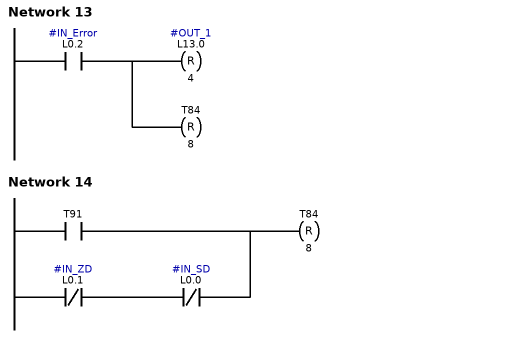
[picture p192: SBR88 networks 13-14]
Network 13
LD     #IN_Error:L0.2
R      #OUT_1:L13.0, 4
R      T84, 8
Network 14
LD     T91
LDN    #IN_ZD:L0.1
AN     #IN_SD:L0.0
OLD
R      T84, 8
END_SUBROUTINE_BLOCK

SUBROUTINE_BLOCK 除铁器4组5:SBR89
TITLE=
VAR_INPUT
IN_SD:BOOL;	// L0.0 
IN_ZD:BOOL;	// L0.1 
IN_Error:BOOL;	// L0.2 
IN_Run_Time:INT;	// LW1 
IN_Stop_Time:INT;	// LW3 
Z_Time:DINT;	// LD5 
END_VAR
VAR_IN_OUT
JS:DINT;	// LD9 
END_VAR
VAR_OUTPUT
OUT_1:BOOL;	// L13.0 
OUT_2:BOOL;	// L13.1 
OUT_3:BOOL;	// L13.2 
OUT_4:BOOL;	// L13.3 
END_VAR
VAR
TP1:BOOL;	// L13.4 
TP2:BOOL;	// L13.5 
END_VAR
BEGIN
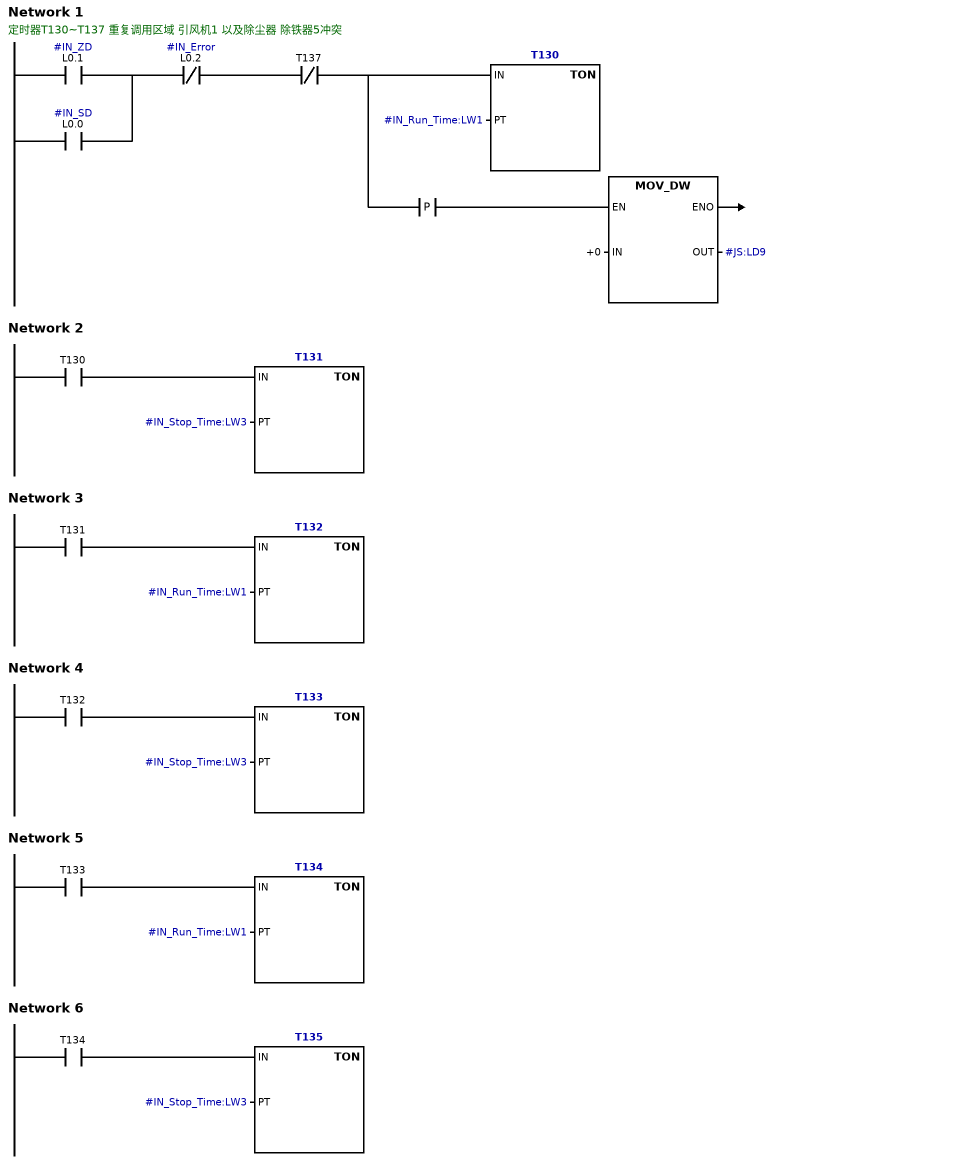
Network 1
// 定时器T130~T137 重复调用区域 引风机1 以及除尘器 除铁器5冲突
LD     #IN_ZD:L0.1
O      #IN_SD:L0.0
AN     #IN_Error:L0.2
AN     T137
TON    T130, #IN_Run_Time:LW1
EU
MOVD   +0, #JS:LD9
Network 2
LD     T130
TON    T131, #IN_Stop_Time:LW3
Network 3
LD     T131
TON    T132, #IN_Run_Time:LW1
Network 4
LD     T132
TON    T133, #IN_Stop_Time:LW3
Network 5
LD     T133
TON    T134, #IN_Run_Time:LW1
Network 6
LD     T134
TON    T135, #IN_Stop_Time:LW3
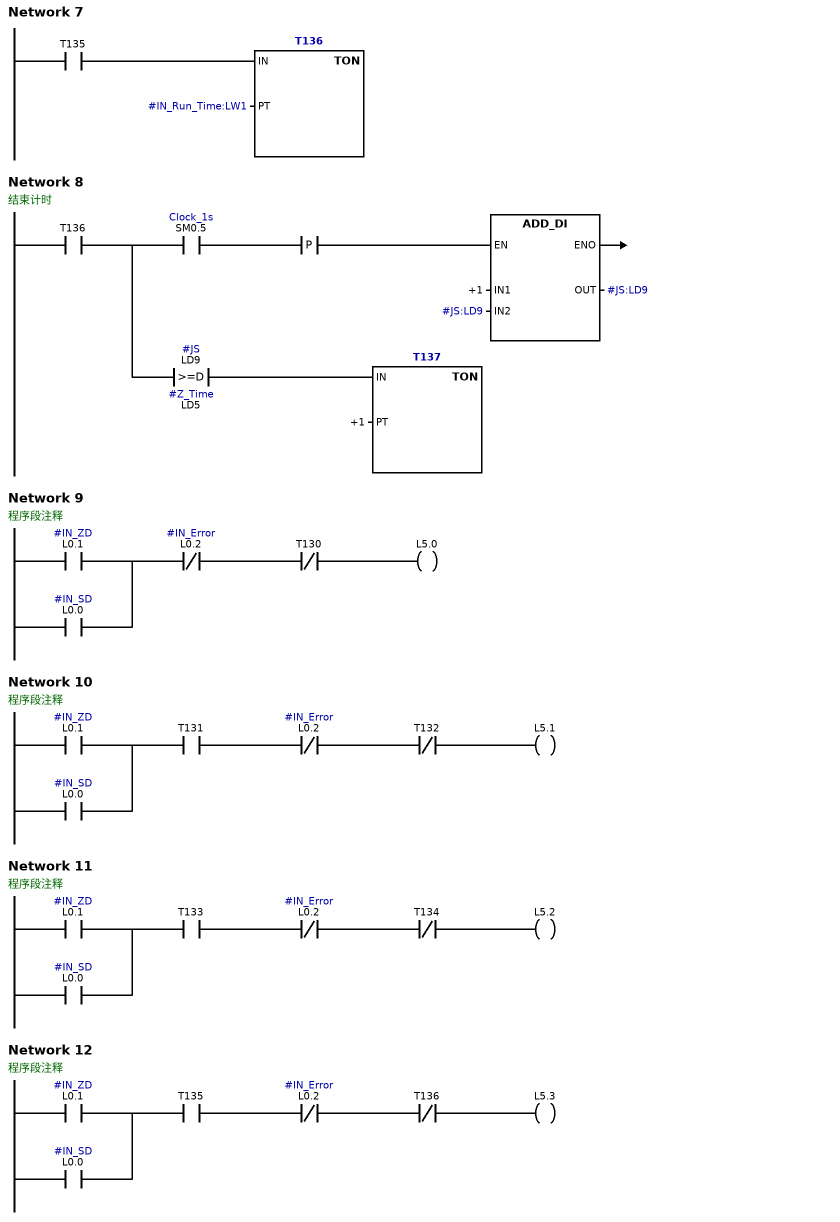
Network 7
LD     T135
TON    T136, #IN_Run_Time:LW1
Network 8
// 结束计时
LD     T136
LPS
A      Clock_1s:SM0.5
EU
+D     +1, #JS:LD9
LPP
AD>=   #JS:LD9, #Z_Time:LD5
TON    T137, +1
Network 9
//  程序段注释
LD     #IN_ZD:L0.1
O      #IN_SD:L0.0
AN     #IN_Error:L0.2
AN     T130
=      L5.0
Network 10
//  程序段注释
LD     #IN_ZD:L0.1
O      #IN_SD:L0.0
A      T131
AN     #IN_Error:L0.2
AN     T132
=      L5.1
Network 11
//  程序段注释
LD     #IN_ZD:L0.1
O      #IN_SD:L0.0
A      T133
AN     #IN_Error:L0.2
AN     T134
=      L5.2
Network 12
//  程序段注释
LD     #IN_ZD:L0.1
O      #IN_SD:L0.0
A      T135
AN     #IN_Error:L0.2
AN     T136
=      L5.3
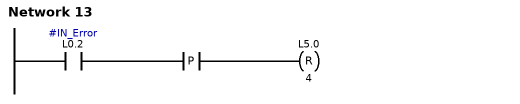
Network 13
LD     #IN_Error:L0.2
EU
R      L5.0, 4
END_SUBROUTINE_BLOCK

SUBROUTINE_BLOCK 膨胀阀4组1:SBR90
TITLE=
VAR_INPUT
IN_SD:BOOL;	// L0.0 
IN_ZD:BOOL;	// L0.1 
IN_Error:BOOL;	// L0.2 
IN_Run_Time:INT;	// LW1 
IN_Stop_Time:INT;	// LW3 
END_VAR
VAR_OUTPUT
OUT_1:BOOL;	// L5.0 膨胀1
OUT_2:BOOL;	// L5.1 下料1
OUT_3:BOOL;	// L5.2 膨胀2
OUT_4:BOOL;	// L5.3 下料2
END_VAR
VAR
TP1:BOOL;	// L5.4 
TP2:BOOL;	// L5.5 
END_VAR
BEGIN
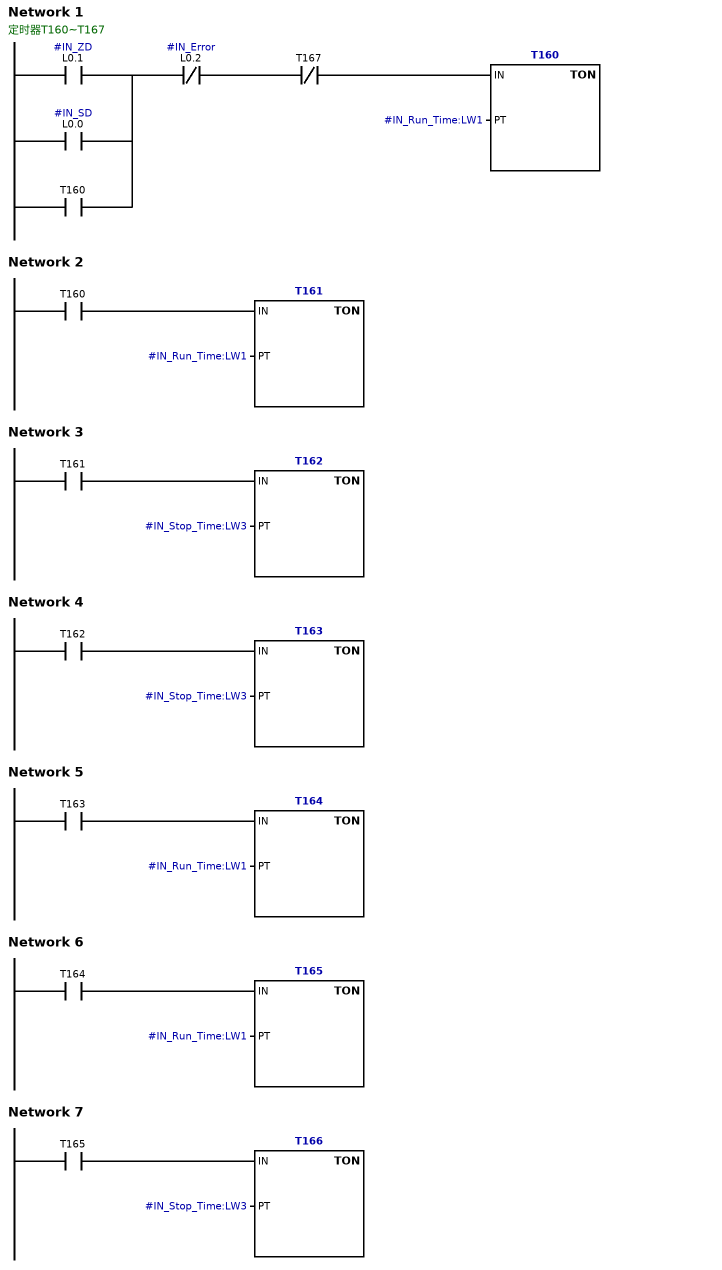
Network 1
// 定时器T160~T167
LD     #IN_ZD:L0.1
O      #IN_SD:L0.0
O      T160
AN     #IN_Error:L0.2
AN     T167
TON    T160, #IN_Run_Time:LW1
Network 2
LD     T160
TON    T161, #IN_Run_Time:LW1
Network 3
LD     T161
TON    T162, #IN_Stop_Time:LW3
Network 4
LD     T162
TON    T163, #IN_Stop_Time:LW3
Network 5
LD     T163
TON    T164, #IN_Run_Time:LW1
Network 6
LD     T164
TON    T165, #IN_Run_Time:LW1
Network 7
LD     T165
TON    T166, #IN_Stop_Time:LW3
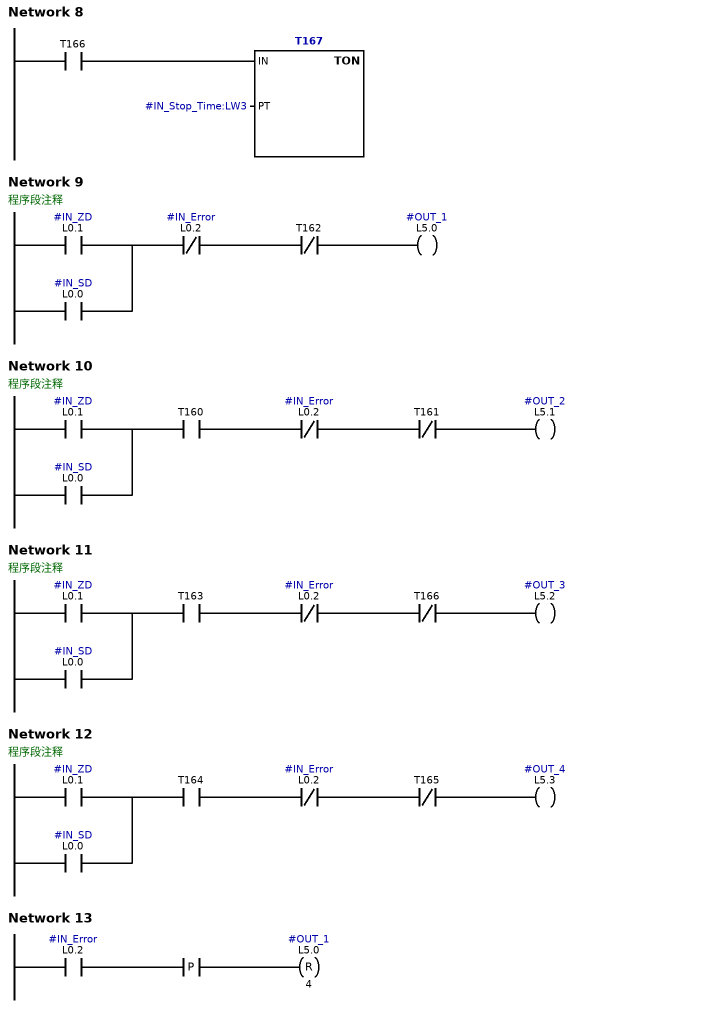
Network 8
LD     T166
TON    T167, #IN_Stop_Time:LW3
Network 9
//  程序段注释
LD     #IN_ZD:L0.1
O      #IN_SD:L0.0
AN     #IN_Error:L0.2
AN     T162
=      #OUT_1:L5.0
Network 10
//  程序段注释
LD     #IN_ZD:L0.1
O      #IN_SD:L0.0
A      T160
AN     #IN_Error:L0.2
AN     T161
=      #OUT_2:L5.1
Network 11
//  程序段注释
LD     #IN_ZD:L0.1
O      #IN_SD:L0.0
A      T163
AN     #IN_Error:L0.2
AN     T166
=      #OUT_3:L5.2
Network 12
//  程序段注释
LD     #IN_ZD:L0.1
O      #IN_SD:L0.0
A      T164
AN     #IN_Error:L0.2
AN     T165
=      #OUT_4:L5.3
Network 13
LD     #IN_Error:L0.2
EU
R      #OUT_1:L5.0, 4
END_SUBROUTINE_BLOCK

SUBROUTINE_BLOCK 膨胀阀4组2:SBR91
TITLE=
VAR_INPUT
IN_SD:BOOL;	// L0.0 
IN_ZD:BOOL;	// L0.1 
IN_Error:BOOL;	// L0.2 
IN_Run_Time:INT;	// LW1 
IN_Stop_Time:INT;	// LW3 
END_VAR
VAR_OUTPUT
OUT_1:BOOL;	// L5.0 
OUT_2:BOOL;	// L5.1 
OUT_3:BOOL;	// L5.2 
OUT_4:BOOL;	// L5.3 
END_VAR
VAR
TP1:BOOL;	// L5.4 
TP2:BOOL;	// L5.5 
END_VAR
BEGIN
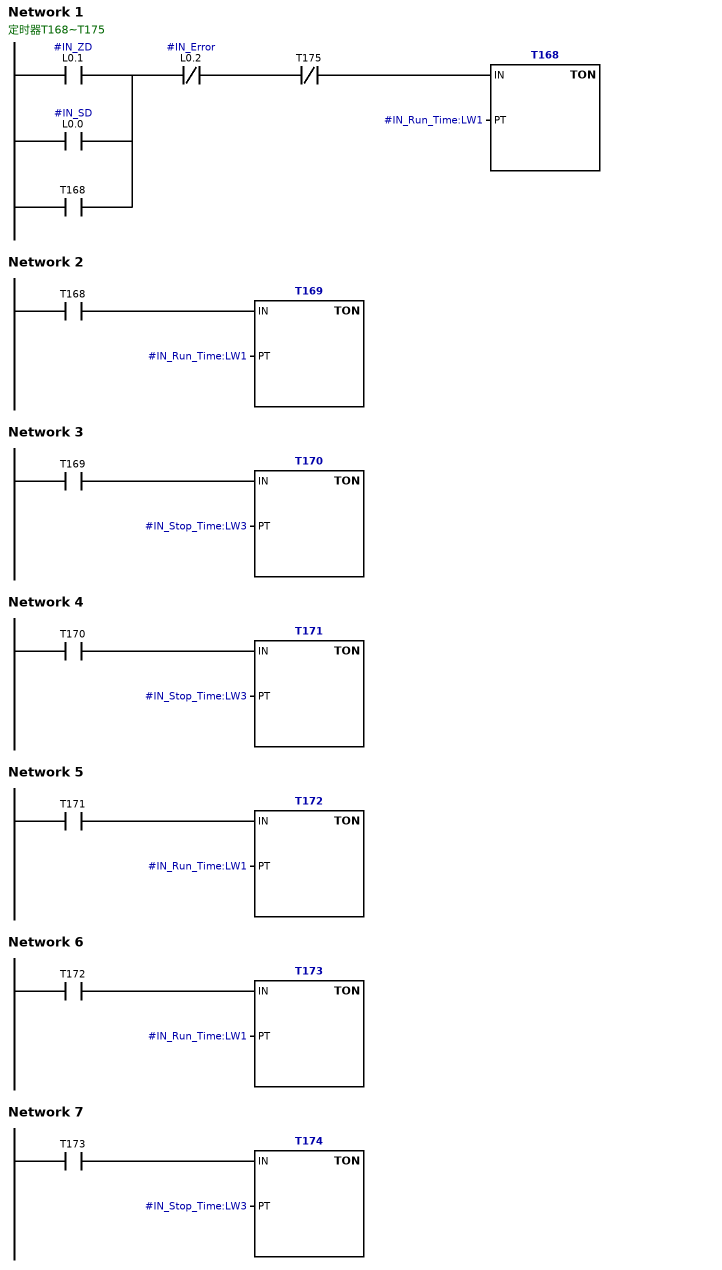
Network 1
// 定时器T168~T175
LD     #IN_ZD:L0.1
O      #IN_SD:L0.0
O      T168
AN     #IN_Error:L0.2
AN     T175
TON    T168, #IN_Run_Time:LW1
Network 2
LD     T168
TON    T169, #IN_Run_Time:LW1
Network 3
LD     T169
TON    T170, #IN_Stop_Time:LW3
Network 4
LD     T170
TON    T171, #IN_Stop_Time:LW3
Network 5
LD     T171
TON    T172, #IN_Run_Time:LW1
Network 6
LD     T172
TON    T173, #IN_Run_Time:LW1
Network 7
LD     T173
TON    T174, #IN_Stop_Time:LW3
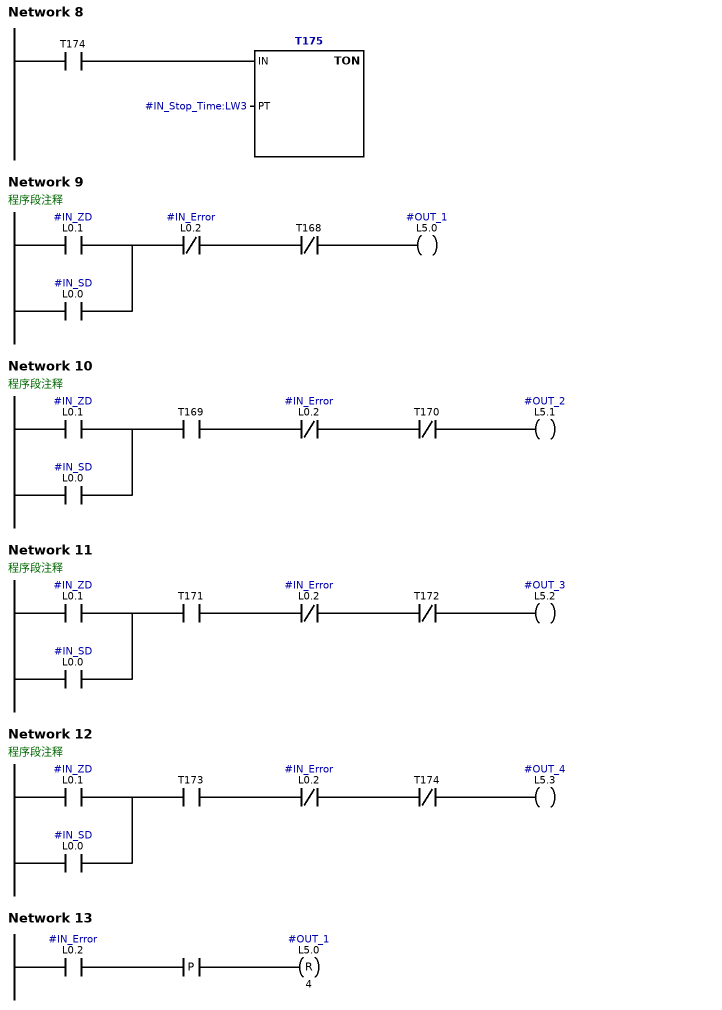
Network 8
LD     T174
TON    T175, #IN_Stop_Time:LW3
Network 9
//  程序段注释
LD     #IN_ZD:L0.1
O      #IN_SD:L0.0
AN     #IN_Error:L0.2
AN     T168
=      #OUT_1:L5.0
Network 10
//  程序段注释
LD     #IN_ZD:L0.1
O      #IN_SD:L0.0
A      T169
AN     #IN_Error:L0.2
AN     T170
=      #OUT_2:L5.1
Network 11
//  程序段注释
LD     #IN_ZD:L0.1
O      #IN_SD:L0.0
A      T171
AN     #IN_Error:L0.2
AN     T172
=      #OUT_3:L5.2
Network 12
//  程序段注释
LD     #IN_ZD:L0.1
O      #IN_SD:L0.0
A      T173
AN     #IN_Error:L0.2
AN     T174
=      #OUT_4:L5.3
Network 13
LD     #IN_Error:L0.2
EU
R      #OUT_1:L5.0, 4
END_SUBROUTINE_BLOCK

SUBROUTINE_BLOCK 膨胀阀4组3:SBR92
TITLE=
VAR_INPUT
IN_SD:BOOL;	// L0.0 
IN_ZD:BOOL;	// L0.1 
IN_Error:BOOL;	// L0.2 
IN_Run_Time:INT;	// LW1 
IN_Stop_Time:INT;	// LW3 
END_VAR
VAR_OUTPUT
OUT_1:BOOL;	// L5.0 
OUT_2:BOOL;	// L5.1 
OUT_3:BOOL;	// L5.2 
OUT_4:BOOL;	// L5.3 
END_VAR
VAR
TP1:BOOL;	// L5.4 
TP2:BOOL;	// L5.5 
END_VAR
BEGIN
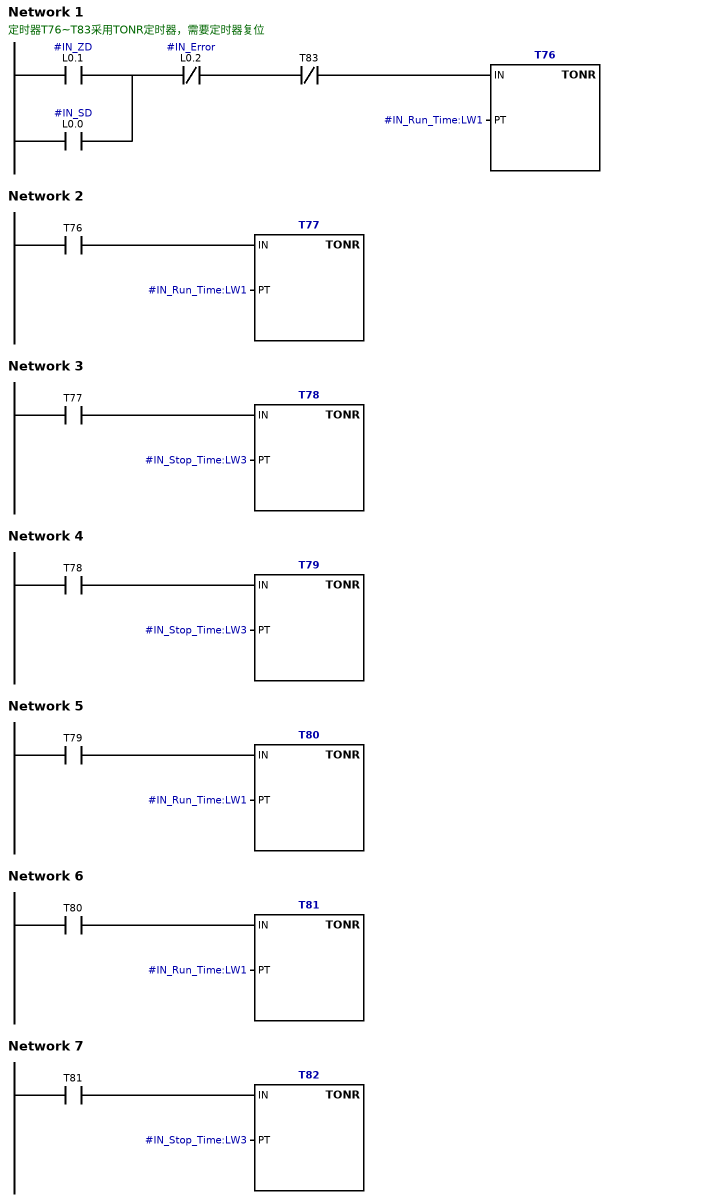
Network 1
// 定时器T76~T83采用TONR定时器，需要定时器复位
LD     #IN_ZD:L0.1
O      #IN_SD:L0.0
AN     #IN_Error:L0.2
AN     T83
TONR   T76, #IN_Run_Time:LW1
Network 2
LD     T76
TONR   T77, #IN_Run_Time:LW1
Network 3
LD     T77
TONR   T78, #IN_Stop_Time:LW3
Network 4
LD     T78
TONR   T79, #IN_Stop_Time:LW3
Network 5
LD     T79
TONR   T80, #IN_Run_Time:LW1
Network 6
LD     T80
TONR   T81, #IN_Run_Time:LW1
Network 7
LD     T81
TONR   T82, #IN_Stop_Time:LW3
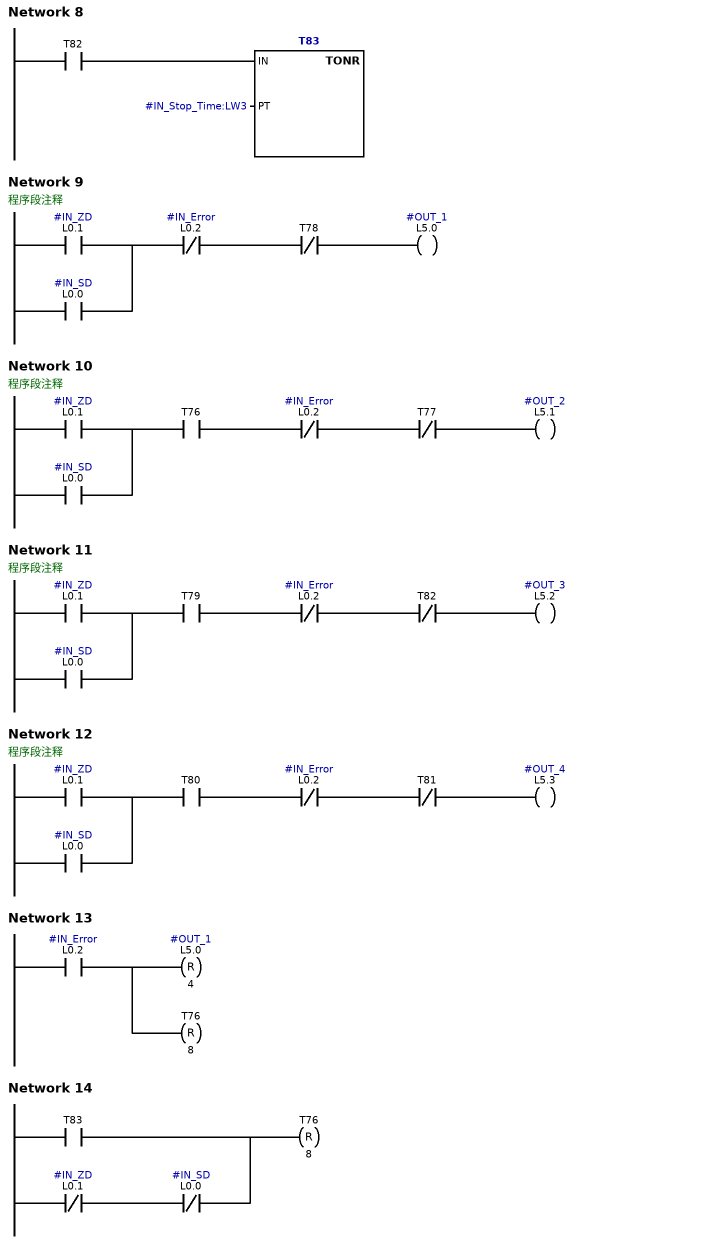
Network 8
LD     T82
TONR   T83, #IN_Stop_Time:LW3
Network 9
//  程序段注释
LD     #IN_ZD:L0.1
O      #IN_SD:L0.0
AN     #IN_Error:L0.2
AN     T78
=      #OUT_1:L5.0
Network 10
//  程序段注释
LD     #IN_ZD:L0.1
O      #IN_SD:L0.0
A      T76
AN     #IN_Error:L0.2
AN     T77
=      #OUT_2:L5.1
Network 11
//  程序段注释
LD     #IN_ZD:L0.1
O      #IN_SD:L0.0
A      T79
AN     #IN_Error:L0.2
AN     T82
=      #OUT_3:L5.2
Network 12
//  程序段注释
LD     #IN_ZD:L0.1
O      #IN_SD:L0.0
A      T80
AN     #IN_Error:L0.2
AN     T81
=      #OUT_4:L5.3
Network 13
LD     #IN_Error:L0.2
R      #OUT_1:L5.0, 4
R      T76, 8
Network 14
LD     T83
LDN    #IN_ZD:L0.1
AN     #IN_SD:L0.0
OLD
R      T76, 8
END_SUBROUTINE_BLOCK

SUBROUTINE_BLOCK 膨胀阀4组4:SBR93
TITLE=
VAR_INPUT
IN_SD:BOOL;	// L0.0 
IN_ZD:BOOL;	// L0.1 
IN_Error:BOOL;	// L0.2 
IN_Run_Time:INT;	// LW1 
IN_Stop_Time:INT;	// LW3 
END_VAR
VAR_OUTPUT
OUT_1:BOOL;	// L5.0 
OUT_2:BOOL;	// L5.1 
OUT_3:BOOL;	// L5.2 
OUT_4:BOOL;	// L5.3 
END_VAR
VAR
TP1:BOOL;	// L5.4 
TP2:BOOL;	// L5.5 
END_VAR
BEGIN
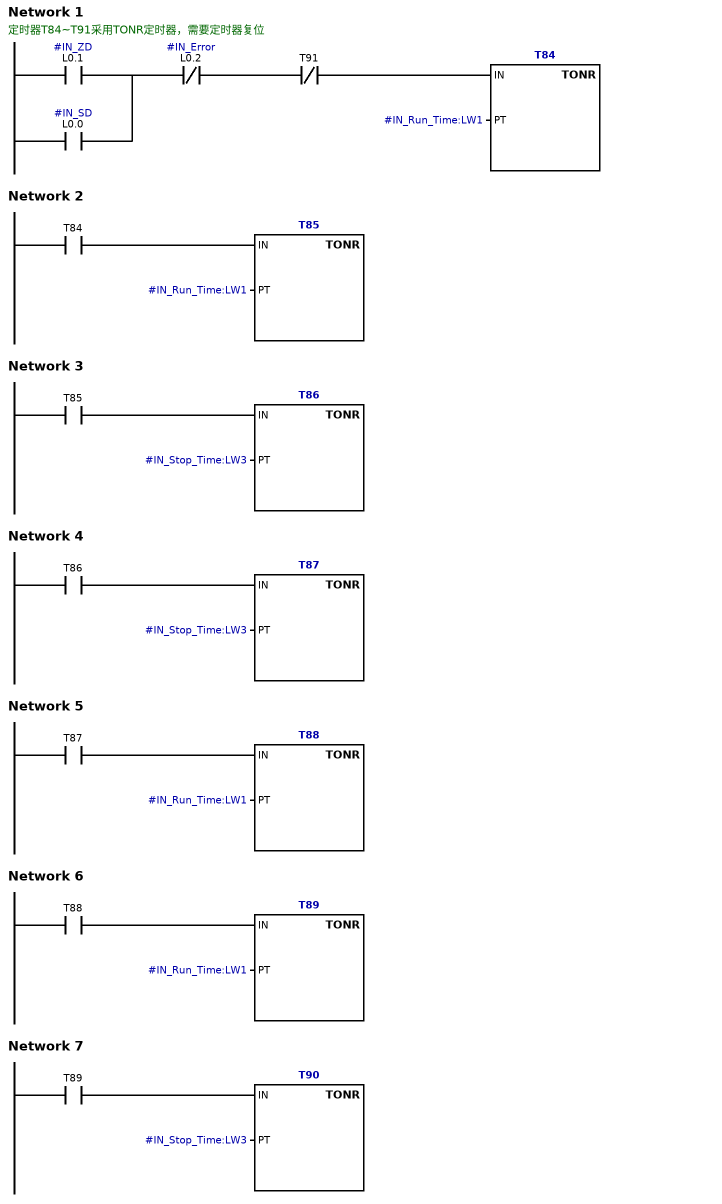
Network 1
// 定时器T84~T91采用TONR定时器，需要定时器复位
LD     #IN_ZD:L0.1
O      #IN_SD:L0.0
AN     #IN_Error:L0.2
AN     T91
TONR   T84, #IN_Run_Time:LW1
Network 2
LD     T84
TONR   T85, #IN_Run_Time:LW1
Network 3
LD     T85
TONR   T86, #IN_Stop_Time:LW3
Network 4
LD     T86
TONR   T87, #IN_Stop_Time:LW3
Network 5
LD     T87
TONR   T88, #IN_Run_Time:LW1
Network 6
LD     T88
TONR   T89, #IN_Run_Time:LW1
Network 7
LD     T89
TONR   T90, #IN_Stop_Time:LW3
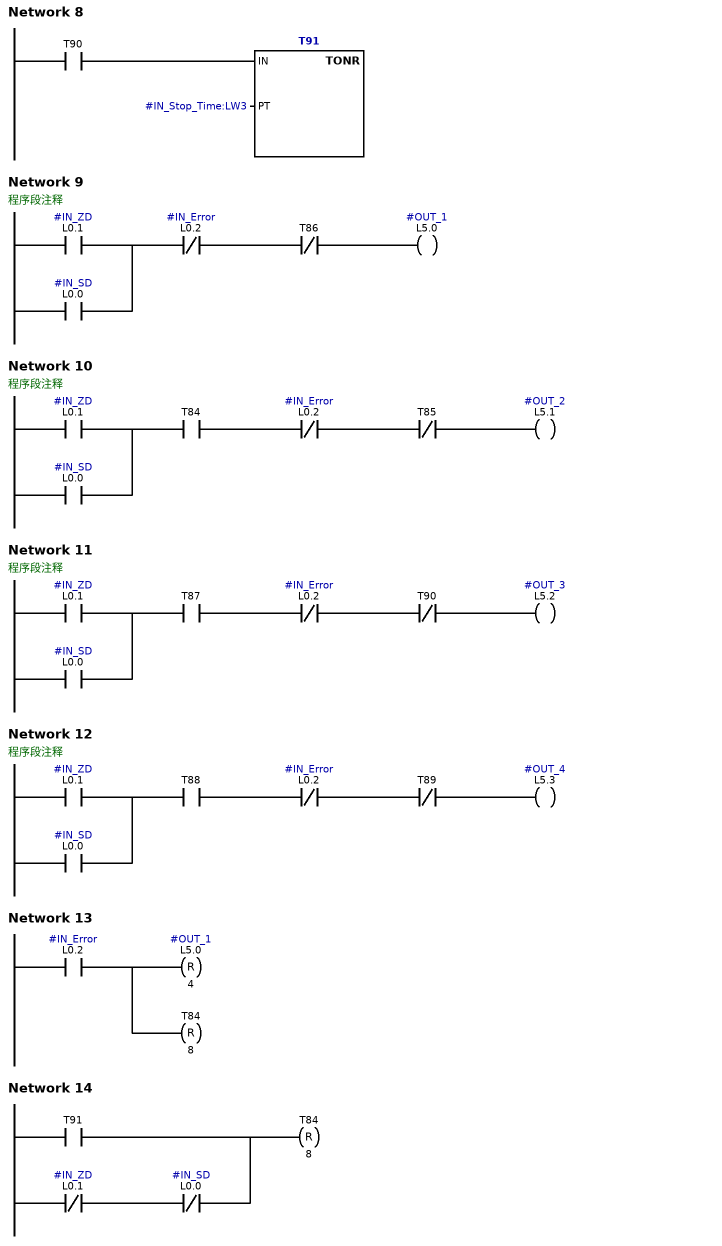
Network 8
LD     T90
TONR   T91, #IN_Stop_Time:LW3
Network 9
//  程序段注释
LD     #IN_ZD:L0.1
O      #IN_SD:L0.0
AN     #IN_Error:L0.2
AN     T86
=      #OUT_1:L5.0
Network 10
//  程序段注释
LD     #IN_ZD:L0.1
O      #IN_SD:L0.0
A      T84
AN     #IN_Error:L0.2
AN     T85
=      #OUT_2:L5.1
Network 11
//  程序段注释
LD     #IN_ZD:L0.1
O      #IN_SD:L0.0
A      T87
AN     #IN_Error:L0.2
AN     T90
=      #OUT_3:L5.2
Network 12
//  程序段注释
LD     #IN_ZD:L0.1
O      #IN_SD:L0.0
A      T88
AN     #IN_Error:L0.2
AN     T89
=      #OUT_4:L5.3
Network 13
LD     #IN_Error:L0.2
R      #OUT_1:L5.0, 4
R      T84, 8
Network 14
LD     T91
LDN    #IN_ZD:L0.1
AN     #IN_SD:L0.0
OLD
R      T84, 8
END_SUBROUTINE_BLOCK

SUBROUTINE_BLOCK Valve1_XH1:SBR100
TITLE=
VAR_INPUT
IN_SD:BOOL;	// L0.0 
IN_ZD:BOOL;	// L0.1 
IN_Error:BOOL;	// L0.2 
IN_Run_Time:INT;	// LW1 
IN_Stop_Time:INT;	// LW3 
END_VAR
VAR_OUTPUT
OUT_ONE:BOOL;	// L5.0 
END_VAR
VAR
TP1:BOOL;	// L5.1 
TP2:BOOL;	// L5.2 
END_VAR
BEGIN
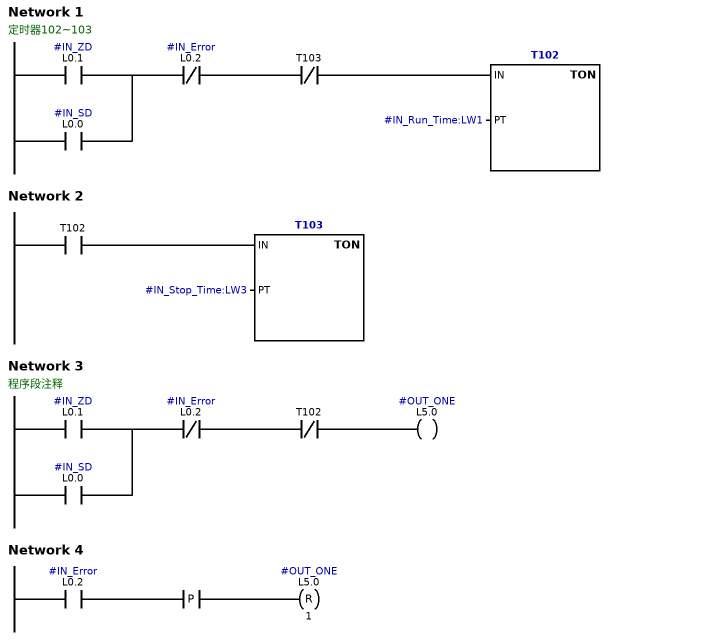
Network 1
// 定时器102~103
LD     #IN_ZD:L0.1
O      #IN_SD:L0.0
AN     #IN_Error:L0.2
AN     T103
TON    T102, #IN_Run_Time:LW1
Network 2
LD     T102
TON    T103, #IN_Stop_Time:LW3
Network 3
// 程序段注释
LD     #IN_ZD:L0.1
O      #IN_SD:L0.0
AN     #IN_Error:L0.2
AN     T102
=      #OUT_ONE:L5.0
Network 4
LD     #IN_Error:L0.2
EU
R      #OUT_ONE:L5.0, 1
END_SUBROUTINE_BLOCK

SUBROUTINE_BLOCK Valve1_XH2:SBR101
TITLE=
VAR_INPUT
IN_SD:BOOL;	// L0.0 
IN_ZD:BOOL;	// L0.1 
IN_Error:BOOL;	// L0.2 
IN_Run_Time:INT;	// LW1 
IN_Stop_Time:INT;	// LW3 
END_VAR
VAR_OUTPUT
OUT_ONE:BOOL;	// L5.0 
END_VAR
VAR
TP1:BOOL;	// L5.1 
TP2:BOOL;	// L5.2 
END_VAR
BEGIN
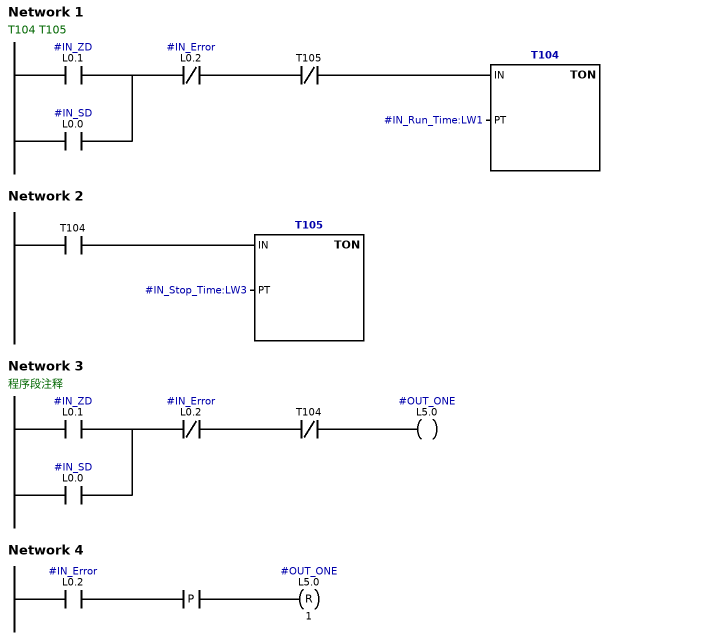
Network 1
// T104 T105
LD     #IN_ZD:L0.1
O      #IN_SD:L0.0
AN     #IN_Error:L0.2
AN     T105
TON    T104, #IN_Run_Time:LW1
Network 2
LD     T104
TON    T105, #IN_Stop_Time:LW3
Network 3
// 程序段注释
LD     #IN_ZD:L0.1
O      #IN_SD:L0.0
AN     #IN_Error:L0.2
AN     T104
=      #OUT_ONE:L5.0
Network 4
LD     #IN_Error:L0.2
EU
R      #OUT_ONE:L5.0, 1
END_SUBROUTINE_BLOCK

SUBROUTINE_BLOCK Valve1_XH3:SBR102
TITLE=
VAR_INPUT
IN_SD:BOOL;	// L0.0 
IN_ZD:BOOL;	// L0.1 
IN_Error:BOOL;	// L0.2 
IN_Run_Time:INT;	// LW1 
IN_Stop_Time:INT;	// LW3 
END_VAR
VAR_OUTPUT
OUT_ONE:BOOL;	// L5.0 
END_VAR
VAR
TP1:BOOL;	// L5.1 
TP2:BOOL;	// L5.2 
END_VAR
BEGIN
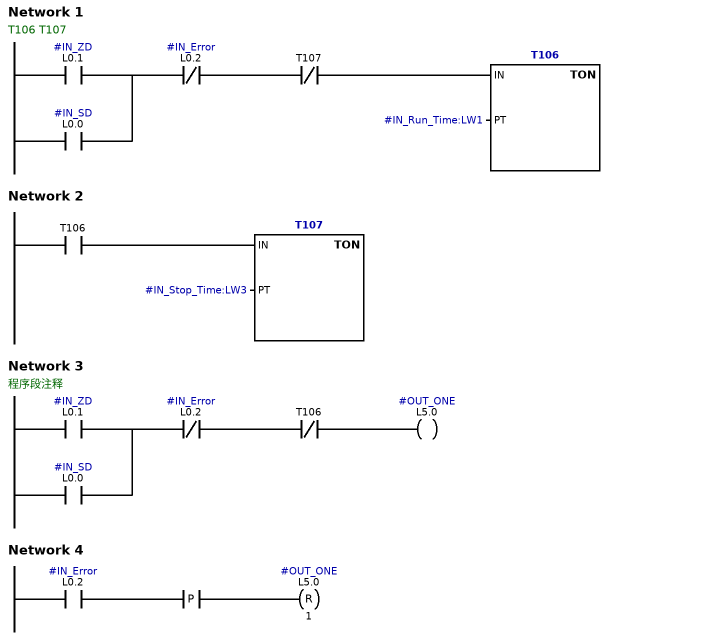
Network 1
// T106 T107
LD     #IN_ZD:L0.1
O      #IN_SD:L0.0
AN     #IN_Error:L0.2
AN     T107
TON    T106, #IN_Run_Time:LW1
Network 2
LD     T106
TON    T107, #IN_Stop_Time:LW3
Network 3
// 程序段注释
LD     #IN_ZD:L0.1
O      #IN_SD:L0.0
AN     #IN_Error:L0.2
AN     T106
=      #OUT_ONE:L5.0
Network 4
LD     #IN_Error:L0.2
EU
R      #OUT_ONE:L5.0, 1
END_SUBROUTINE_BLOCK

SUBROUTINE_BLOCK Valve1_XH4:SBR103
TITLE=
VAR_INPUT
IN_SD:BOOL;	// L0.0 
IN_ZD:BOOL;	// L0.1 
IN_Error:BOOL;	// L0.2 
IN_Run_Time:INT;	// LW1 
IN_Stop_Time:INT;	// LW3 
END_VAR
VAR_OUTPUT
OUT_ONE:BOOL;	// L5.0 
END_VAR
VAR
TP1:BOOL;	// L5.1 
TP2:BOOL;	// L5.2 
END_VAR
BEGIN
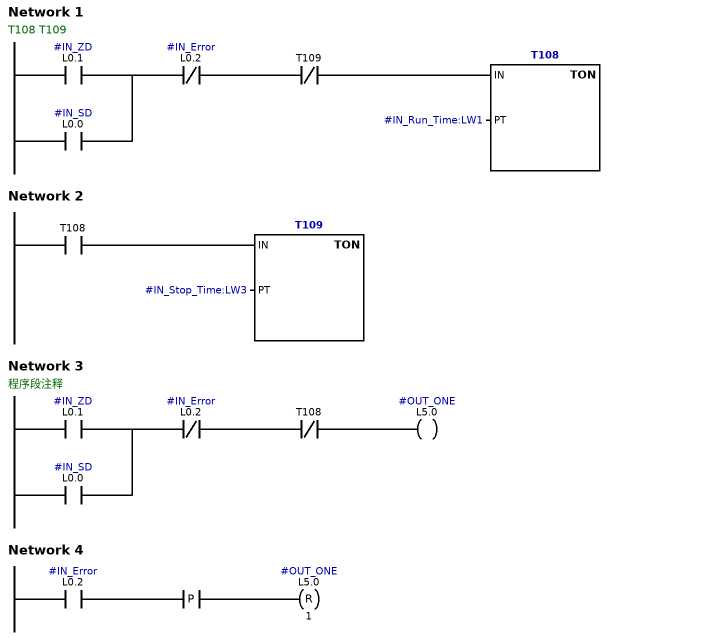
Network 1
// T108 T109
LD     #IN_ZD:L0.1
O      #IN_SD:L0.0
AN     #IN_Error:L0.2
AN     T109
TON    T108, #IN_Run_Time:LW1
Network 2
LD     T108
TON    T109, #IN_Stop_Time:LW3
Network 3
// 程序段注释
LD     #IN_ZD:L0.1
O      #IN_SD:L0.0
AN     #IN_Error:L0.2
AN     T108
=      #OUT_ONE:L5.0
Network 4
LD     #IN_Error:L0.2
EU
R      #OUT_ONE:L5.0, 1
END_SUBROUTINE_BLOCK

SUBROUTINE_BLOCK Valve1_XH5:SBR104
TITLE=
VAR_INPUT
IN_SD:BOOL;	// L0.0 
IN_ZD:BOOL;	// L0.1 
IN_Error:BOOL;	// L0.2 
IN_Run_Time:INT;	// LW1 
IN_Stop_Time:INT;	// LW3 
END_VAR
VAR_OUTPUT
OUT_ONE:BOOL;	// L5.0 
END_VAR
VAR
TP1:BOOL;	// L5.1 
TP2:BOOL;	// L5.2 
END_VAR
BEGIN
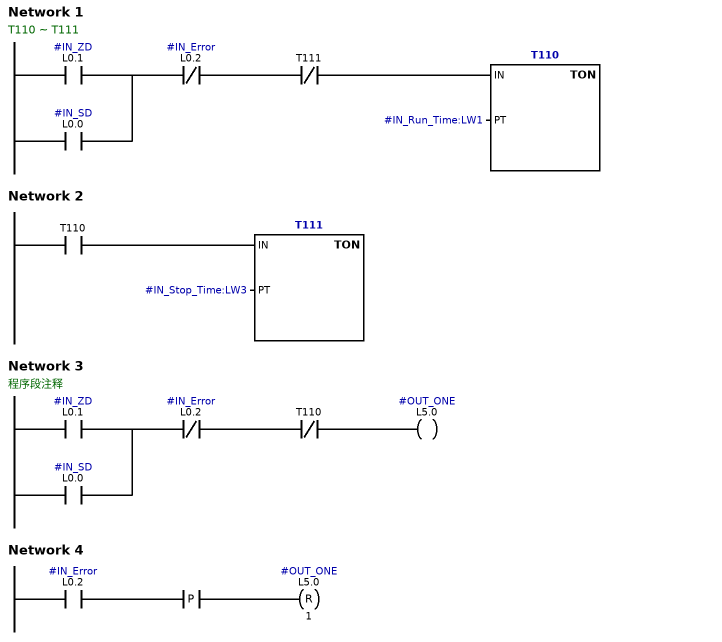
Network 1
// T110 ~ T111
LD     #IN_ZD:L0.1
O      #IN_SD:L0.0
AN     #IN_Error:L0.2
AN     T111
TON    T110, #IN_Run_Time:LW1
Network 2
LD     T110
TON    T111, #IN_Stop_Time:LW3
Network 3
// 程序段注释
LD     #IN_ZD:L0.1
O      #IN_SD:L0.0
AN     #IN_Error:L0.2
AN     T110
=      #OUT_ONE:L5.0
Network 4
LD     #IN_Error:L0.2
EU
R      #OUT_ONE:L5.0, 1
END_SUBROUTINE_BLOCK

SUBROUTINE_BLOCK Valve1_XH6:SBR105
TITLE=
VAR_INPUT
IN_SD:BOOL;	// L0.0 
IN_ZD:BOOL;	// L0.1 
IN_Error:BOOL;	// L0.2 
IN_Run_Time:INT;	// LW1 
IN_Stop_Time:INT;	// LW3 
END_VAR
VAR_OUTPUT
OUT_ONE:BOOL;	// L5.0 
END_VAR
VAR
TP1:BOOL;	// L5.1 
TP2:BOOL;	// L5.2 
END_VAR
BEGIN
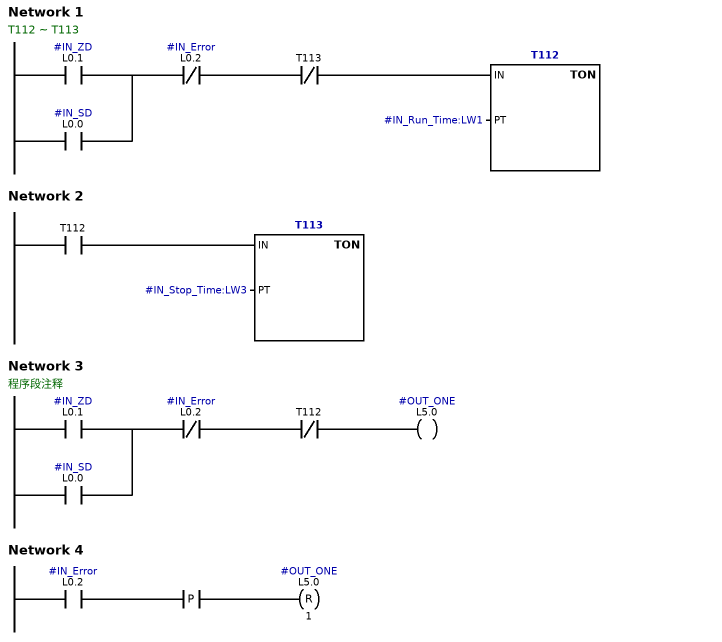
Network 1
// T112 ~ T113
LD     #IN_ZD:L0.1
O      #IN_SD:L0.0
AN     #IN_Error:L0.2
AN     T113
TON    T112, #IN_Run_Time:LW1
Network 2
LD     T112
TON    T113, #IN_Stop_Time:LW3
Network 3
// 程序段注释
LD     #IN_ZD:L0.1
O      #IN_SD:L0.0
AN     #IN_Error:L0.2
AN     T112
=      #OUT_ONE:L5.0
Network 4
LD     #IN_Error:L0.2
EU
R      #OUT_ONE:L5.0, 1
END_SUBROUTINE_BLOCK

SUBROUTINE_BLOCK Valve1_XH7:SBR106
TITLE=
VAR_INPUT
IN_SD:BOOL;	// L0.0 
IN_ZD:BOOL;	// L0.1 
IN_Error:BOOL;	// L0.2 
IN_Run_Time:INT;	// LW1 
IN_Stop_Time:INT;	// LW3 
END_VAR
VAR_OUTPUT
OUT_ONE:BOOL;	// L5.0 
END_VAR
VAR
TP1:BOOL;	// L5.1 
TP2:BOOL;	// L5.2 
END_VAR
BEGIN
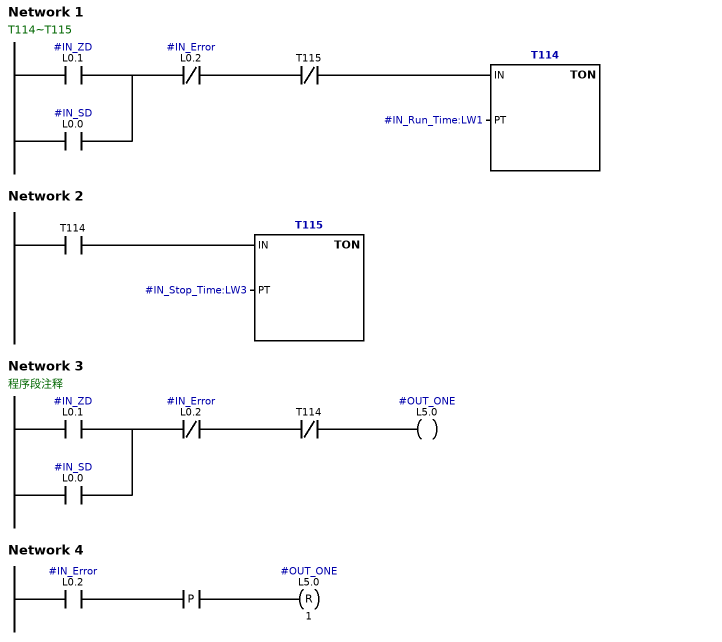
Network 1
// T114~T115
LD     #IN_ZD:L0.1
O      #IN_SD:L0.0
AN     #IN_Error:L0.2
AN     T115
TON    T114, #IN_Run_Time:LW1
Network 2
LD     T114
TON    T115, #IN_Stop_Time:LW3
Network 3
// 程序段注释
LD     #IN_ZD:L0.1
O      #IN_SD:L0.0
AN     #IN_Error:L0.2
AN     T114
=      #OUT_ONE:L5.0
Network 4
LD     #IN_Error:L0.2
EU
R      #OUT_ONE:L5.0, 1
END_SUBROUTINE_BLOCK

SUBROUTINE_BLOCK Valve1_XH8:SBR107
TITLE=
VAR_INPUT
IN_SD:BOOL;	// L0.0 
IN_ZD:BOOL;	// L0.1 
IN_Error:BOOL;	// L0.2 
IN_Run_Time:INT;	// LW1 
IN_Stop_Time:INT;	// LW3 
END_VAR
VAR_OUTPUT
OUT_ONE:BOOL;	// L5.0 
END_VAR
VAR
TP1:BOOL;	// L5.1 
TP2:BOOL;	// L5.2 
END_VAR
BEGIN
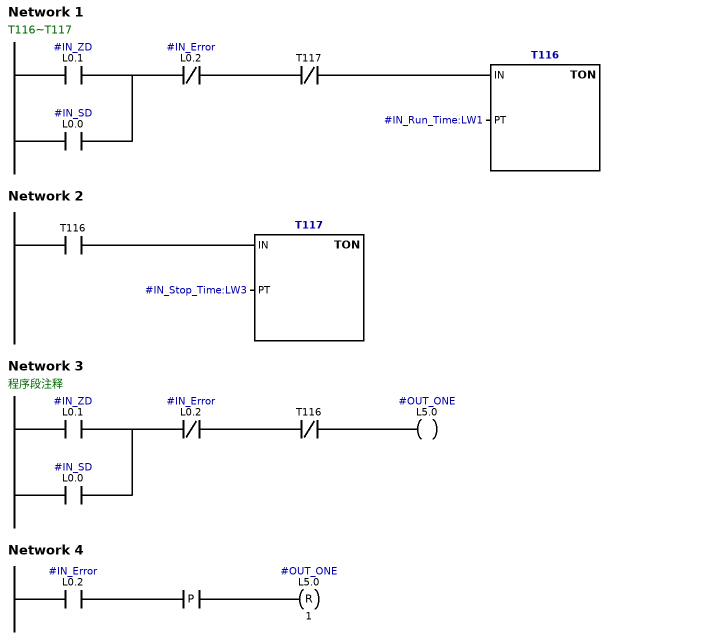
Network 1
// T116~T117
LD     #IN_ZD:L0.1
O      #IN_SD:L0.0
AN     #IN_Error:L0.2
AN     T117
TON    T116, #IN_Run_Time:LW1
Network 2
LD     T116
TON    T117, #IN_Stop_Time:LW3
Network 3
// 程序段注释
LD     #IN_ZD:L0.1
O      #IN_SD:L0.0
AN     #IN_Error:L0.2
AN     T116
=      #OUT_ONE:L5.0
Network 4
LD     #IN_Error:L0.2
EU
R      #OUT_ONE:L5.0, 1
END_SUBROUTINE_BLOCK

SUBROUTINE_BLOCK Valve1_XH9:SBR108
TITLE=
VAR_INPUT
IN_SD:BOOL;	// L0.0 
IN_ZD:BOOL;	// L0.1 
IN_Error:BOOL;	// L0.2 
IN_Run_Time:INT;	// LW1 
IN_Stop_Time:INT;	// LW3 
END_VAR
VAR_OUTPUT
OUT_ONE:BOOL;	// L5.0 
END_VAR
VAR
TP1:BOOL;	// L5.1 
TP2:BOOL;	// L5.2 
END_VAR
BEGIN
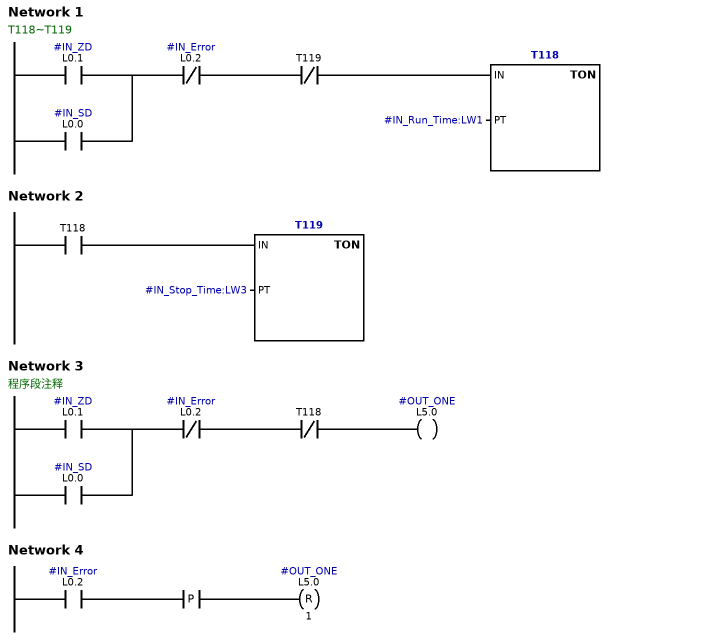
Network 1
// T118~T119
LD     #IN_ZD:L0.1
O      #IN_SD:L0.0
AN     #IN_Error:L0.2
AN     T119
TON    T118, #IN_Run_Time:LW1
Network 2
LD     T118
TON    T119, #IN_Stop_Time:LW3
Network 3
// 程序段注释
LD     #IN_ZD:L0.1
O      #IN_SD:L0.0
AN     #IN_Error:L0.2
AN     T118
=      #OUT_ONE:L5.0
Network 4
LD     #IN_Error:L0.2
EU
R      #OUT_ONE:L5.0, 1
END_SUBROUTINE_BLOCK

SUBROUTINE_BLOCK Valve1_XH10:SBR109
TITLE=
VAR_INPUT
IN_SD:BOOL;	// L0.0 
IN_ZD:BOOL;	// L0.1 
IN_Error:BOOL;	// L0.2 
IN_Run_Time:INT;	// LW1 
IN_Stop_Time:INT;	// LW3 
END_VAR
VAR_OUTPUT
OUT_ONE:BOOL;	// L5.0 
END_VAR
VAR
TP1:BOOL;	// L5.1 
TP2:BOOL;	// L5.2 
END_VAR
BEGIN
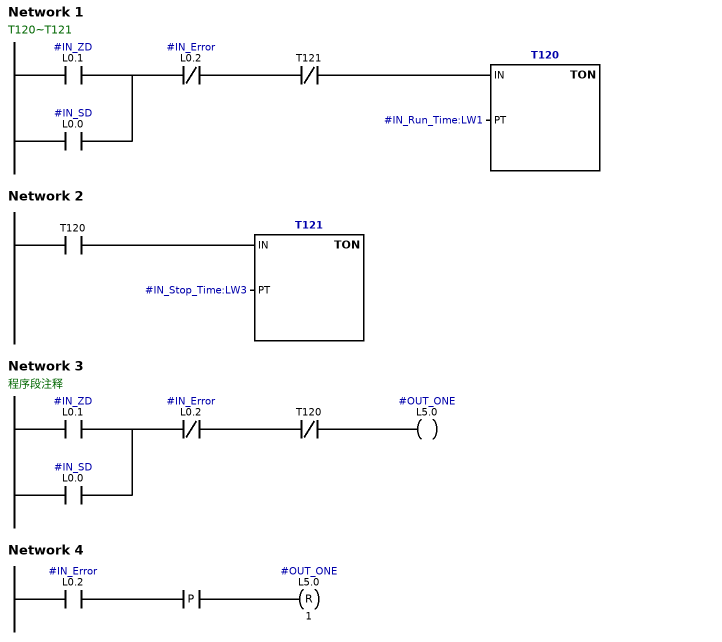
Network 1
// T120~T121
LD     #IN_ZD:L0.1
O      #IN_SD:L0.0
AN     #IN_Error:L0.2
AN     T121
TON    T120, #IN_Run_Time:LW1
Network 2
LD     T120
TON    T121, #IN_Stop_Time:LW3
Network 3
// 程序段注释
LD     #IN_ZD:L0.1
O      #IN_SD:L0.0
AN     #IN_Error:L0.2
AN     T120
=      #OUT_ONE:L5.0
Network 4
LD     #IN_Error:L0.2
EU
R      #OUT_ONE:L5.0, 1
END_SUBROUTINE_BLOCK

SUBROUTINE_BLOCK Valve1_XH11:SBR110
TITLE=
VAR_INPUT
IN_SD:BOOL;	// L0.0 
IN_ZD:BOOL;	// L0.1 
IN_Error:BOOL;	// L0.2 
IN_Run_Time:INT;	// LW1 
IN_Stop_Time:INT;	// LW3 
END_VAR
VAR_OUTPUT
OUT_ONE:BOOL;	// L5.0 
END_VAR
VAR
TP1:BOOL;	// L5.1 
TP2:BOOL;	// L5.2 
END_VAR
BEGIN
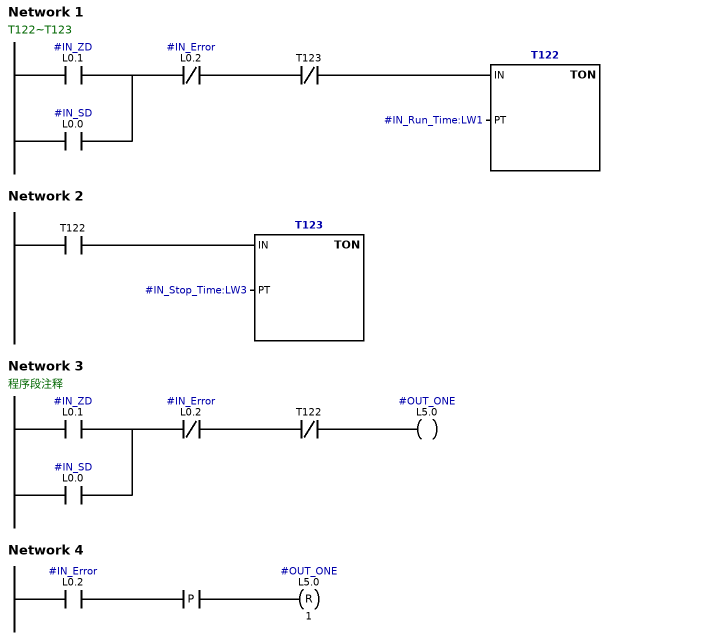
Network 1
// T122~T123
LD     #IN_ZD:L0.1
O      #IN_SD:L0.0
AN     #IN_Error:L0.2
AN     T123
TON    T122, #IN_Run_Time:LW1
Network 2
LD     T122
TON    T123, #IN_Stop_Time:LW3
Network 3
// 程序段注释
LD     #IN_ZD:L0.1
O      #IN_SD:L0.0
AN     #IN_Error:L0.2
AN     T122
=      #OUT_ONE:L5.0
Network 4
LD     #IN_Error:L0.2
EU
R      #OUT_ONE:L5.0, 1
END_SUBROUTINE_BLOCK

SUBROUTINE_BLOCK Valve1_XH12:SBR111
TITLE=
VAR_INPUT
IN_SD:BOOL;	// L0.0 
IN_ZD:BOOL;	// L0.1 
IN_Error:BOOL;	// L0.2 
IN_Run_Time:INT;	// LW1 
IN_Stop_Time:INT;	// LW3 
END_VAR
VAR_OUTPUT
OUT_ONE:BOOL;	// L5.0 
END_VAR
VAR
TP1:BOOL;	// L5.1 
TP2:BOOL;	// L5.2 
END_VAR
BEGIN
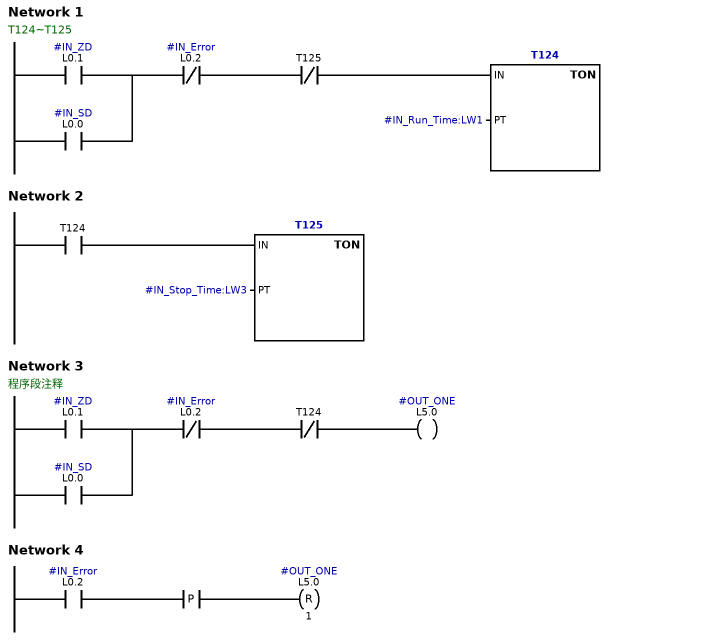
Network 1
// T124~T125
LD     #IN_ZD:L0.1
O      #IN_SD:L0.0
AN     #IN_Error:L0.2
AN     T125
TON    T124, #IN_Run_Time:LW1
Network 2
LD     T124
TON    T125, #IN_Stop_Time:LW3
Network 3
// 程序段注释
LD     #IN_ZD:L0.1
O      #IN_SD:L0.0
AN     #IN_Error:L0.2
AN     T124
=      #OUT_ONE:L5.0
Network 4
LD     #IN_Error:L0.2
EU
R      #OUT_ONE:L5.0, 1
END_SUBROUTINE_BLOCK

SUBROUTINE_BLOCK Valve1_XH13:SBR112
TITLE=
VAR_INPUT
IN_SD:BOOL;	// L0.0 
IN_ZD:BOOL;	// L0.1 
IN_Error:BOOL;	// L0.2 
IN_Run_Time:INT;	// LW1 
IN_Stop_Time:INT;	// LW3 
END_VAR
VAR_OUTPUT
OUT_ONE:BOOL;	// L5.0 
END_VAR
VAR
TP1:BOOL;	// L5.1 
TP2:BOOL;	// L5.2 
END_VAR
BEGIN
